TYPE ST_MachinePermissions :
STRUCT
	(* REZERWA *)
	bPermission00 : BOOL;
	(* REZERWA *)
	bPermission01 : BOOL;
	(* REZERWA *)
	bPermission02 : BOOL;
	(* REZERWA *)
	bPermission03 : BOOL;
	(* REZERWA *)
	bPermission04 : BOOL;
	(* REZERWA *)
	bPermission05 : BOOL;
	(* REZERWA *)
	bPermission06 : BOOL;
	(* REZERWA *)
	bPermission07 : BOOL;
	(* REZERWA *)
	bPermission10 : BOOL;
	(* REZERWA *)
	bPermission11 : BOOL;
	(* REZERWA *)
	bPermission12 : BOOL;
	(* REZERWA *)
	bPermission13 : BOOL;
	(* REZERWA *)
	bPermission14 : BOOL;
	(* REZERWA *)
	bPermission15 : BOOL;
	(* REZERWA *)
	bPermission16 : BOOL;
	(* REZERWA *)
	bPermission17 : BOOL;
END_STRUCT
END_TYPE

(* stored: Version 1.1.0.1, ProductVersion 3.1.4026.13, FileIdentifier 57d4eb0e337e5c687ec09d8c473c1baa232add80, FileSignature 787635bee9a96ae003060904b8916c03c05bdb9a79ddd71d2359117bac555f6c1cbd6b47eaa2847df32dea263c298f465e2a186c109e98a7d1ef2806b32008a1a2715ad1ca79265990e421abb3ef16d2ab62198d843fd4c11b742d09cec0da660729853a3dfde1842ad9ec23726dba9c21c1b09addb427ed9e764e597a1f62986556057dabf5d0332c862715dc3710c5840c5ef05d59f6aaa9c87e5a4eac3ee0c3c3c36329d9af2ac1568709d31f65eab1e7dc1a96559e6fa94efc69d75bd4d5a8e3dc77d72e12d94605a7f1d78e4030073e94e5c78914c0ee699cc1b2ea12e6c7b7ef82d6a917542ce191b9167639a7b2819e73bae8a09ace2715ee318e5a60
   DUT ST_MachinePermissions: Id {0a5a9340-871f-4434-84f8-67ba0c96138c} *)
